FUNCTION_BLOCK PUBLIC TestEcatComponent EXTENDS TcoIo.TcoEcatComponent

VAR_OUTPUT
END_VAR
VAR
END_VAR

SUPER^(AdsAddr:= AdsAddr);

END_FUNCTION_BLOCK

(* stored: Version 1.1.0.1, ProductVersion 3.1.4024.10
   POU TestEcatComponent: Id {ce615717-6db6-0331-2bc3-c8a98ad8d687}, SpecialFunc None *)
